RoboDK station: container_v08.rdk

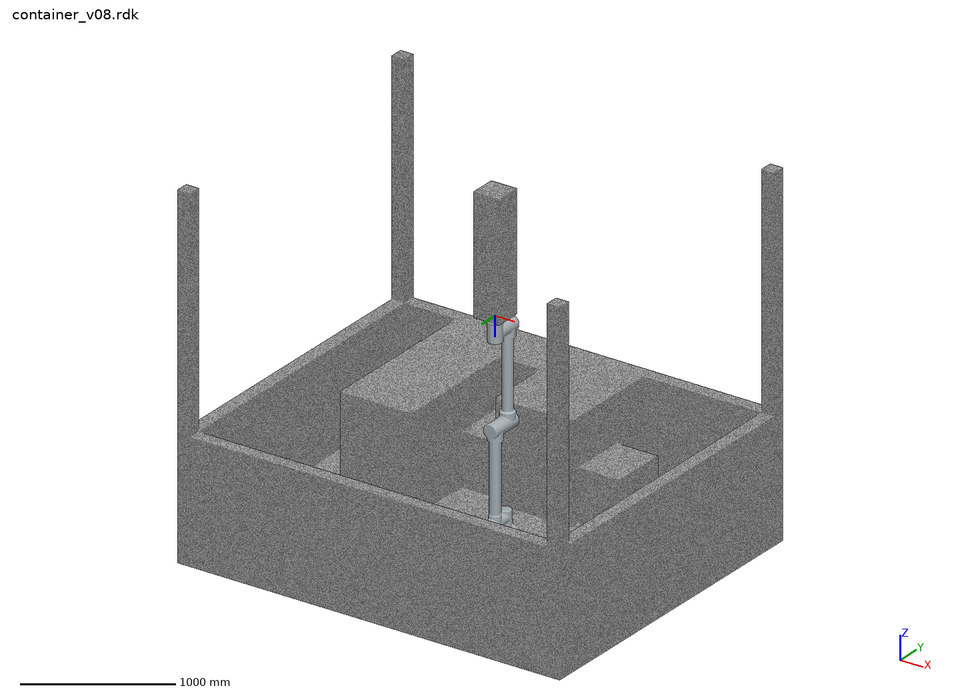
[picture v0: the station drawn from its stored meshes, robots at their saved joint values, targets as dots, program paths as lines]
Station container_v08 (saved by RoboDK 5.4.0). Poses are relative to the parent item; angles as X-Y-Z fixed-axis rotations.
  - frame Avena arm Base at (607.5, -10, 1600) mm, rotated rx 180 ry 0 rz 0 deg
    - robot Avena arm: 6 axes
        modified DH rows (alpha deg, a mm, theta deg, d mm): 0, 0, 0, 123.3; 90, 0, 90, 0; 0, 686, 0, 0; 0, 671, -90, 116.4; -90, 0, 0, 115.4; 90, 0, 0, 67.4
        joint limits [-174.7, -90, -166, -174.7, -174.7, -174.7] to [174.7, 90, 166, 174.7, 174.7, 174.7]; home [0, 0, 0, 0, 0, 0]; saved at [0, 0, 0, 0, 0, 0]
  - object kontener v08 stp at (0, 0, 0) mm, size 3000 x 2500 x 2665 mm, geometry from kontener v08 stp.stp
